FUNCTION_BLOCK FB_GuidanceSystem IMPLEMENTS ITF_HighLevelSystem
VAR_INPUT
	eState : GuidanceSystemSTM;
END_VAR
VAR
	fbAccelerationSensor1 : FB_AccelerationSensor;
	fbAccelerationSensor2 : FB_AccelerationSensor;
	fbGuidanceControllerXMC1 : FB_GuidanceController;
	fbGuidanceControllerXMC2 : FB_GuidanceController;
	fbGuidanceControllerXMC3 : FB_GuidanceController;
	fbGuidanceControllerXMC4 : FB_GuidanceController;
END_VAR

IF eActivationStatus = ActivationStatus.Enabled THEN
	//High Level State Machine
	CASE eState OF
		GuidanceSystemSTM.Idling:
				bEnableCurrentController := FALSE;		

				fbGuidanceControllerXMC1.bActive := FALSE;
				fbGuidanceControllerXMC2.bActive := FALSE;
				fbGuidanceControllerXMC3.bActive := FALSE;
				fbGuidanceControllerXMC4.bActive := FALSE;
		
				fbAccelerationSensor1();
				fbAccelerationSensor2();
				fbGuidanceControllerXMC1();
				fbGuidanceControllerXMC2();
				fbGuidanceControllerXMC3();
				fbGuidanceControllerXMC4();	
		
		
		GuidanceSystemSTM.PreRunning:
				bEnableCurrentController := FALSE;		

				fbAccelerationSensor1();
				fbAccelerationSensor2();
				fbGuidanceControllerXMC1();
				fbGuidanceControllerXMC2();
				fbGuidanceControllerXMC3();
				fbGuidanceControllerXMC4();	
		
		
		GuidanceSystemSTM.Running:
				bEnableCurrentController := TRUE;
		
				fbGuidanceControllerXMC1.bActive := TRUE;
				fbGuidanceControllerXMC2.bActive := TRUE;
				fbGuidanceControllerXMC3.bActive := TRUE;
				fbGuidanceControllerXMC4.bActive := TRUE;

				fbAccelerationSensor1();
				fbAccelerationSensor2();
				fbGuidanceControllerXMC1();
				fbGuidanceControllerXMC2();
				fbGuidanceControllerXMC3();
				fbGuidanceControllerXMC4();		

		GuidanceSystemSTM.PostRunning:
				bEnableCurrentController := FALSE;
		
				fbGuidanceControllerXMC1.bActive := FALSE;
				fbGuidanceControllerXMC2.bActive := FALSE;
				fbGuidanceControllerXMC3.bActive := FALSE;
				fbGuidanceControllerXMC4.bActive := FALSE;
				
				fbAccelerationSensor1();
				fbAccelerationSensor2();
				fbGuidanceControllerXMC1();
				fbGuidanceControllerXMC2();
				fbGuidanceControllerXMC3();
				fbGuidanceControllerXMC4();			
	END_CASE
END_IF

PROPERTY aIMU1Acceleration : ARRAY [0..2] OF REAL
GET
aIMU1Acceleration := fbAccelerationSensor1.aAccelerationValues;
END_GET
END_PROPERTY

PROPERTY aIMU2Acceleration : ARRAY [0..2] OF REAL
GET
aIMU2Acceleration := fbAccelerationSensor1.aAccelerationValues;
END_GET
END_PROPERTY

PROPERTY PUBLIC bEnableCurrentController : BOOL
GET
END_GET
SET // PUBLIC
fbGuidanceControllerXMC1.bActive := bEnableCurrentController;
fbGuidanceControllerXMC2.bActive := bEnableCurrentController;
fbGuidanceControllerXMC3.bActive := bEnableCurrentController;
fbGuidanceControllerXMC4.bActive := bEnableCurrentController;
END_SET
END_PROPERTY

PROPERTY PUBLIC bEnableIControl : BOOL
GET
VAR
	nControlOption : USINT;
END_VAR
nControlOption := nGCControlOption;

IF nControlOption.0 THEN
	bEnableIControl := TRUE;
ELSE
	bEnableIControl := FALSE;
END_IF
END_GET
END_PROPERTY

PROPERTY PUBLIC bEnablePControl : BOOL
GET
VAR
	nControlOption : USINT;
END_VAR
nControlOption := nGCControlOption;

IF nControlOption.1 THEN
	bEnablePControl := TRUE;
ELSE
	bEnablePControl := FALSE;
END_IF
END_GET
END_PROPERTY

PROPERTY eActivationStatus : ActivationStatus
GET
END_GET
SET
END_SET
END_PROPERTY

PROPERTY eCondition : HighLevelCondition
GET
IF eActivationStatus = ActivationStatus.Disabled THEN
	eCondition := HighLevelCondition.SLEEP;
ELSE
	IF fbAccelerationSensor1.eCondition = SubLevelCondition.RUN AND fbAccelerationSensor2.eCondition = SubLevelCondition.RUN AND fbGuidanceController.eCondition = SubLevelCondition.RUN THEN
		eCondition := HighLevelCondition.RUN;
	ELSE
		eCondition := HighLevelCondition.INIT;
	END_IF
END_IF
END_GET
END_PROPERTY

PROPERTY PUBLIC eGCOperationMode : BOOL
SET
IF NOT eGCOperationMode THEN
	fbGuidanceControllerXMC1.eOperationMode := GuidanceControllerOperationMode.CurrentControlled;
	fbGuidanceControllerXMC2.eOperationMode := GuidanceControllerOperationMode.CurrentControlled;
	fbGuidanceControllerXMC3.eOperationMode := GuidanceControllerOperationMode.CurrentControlled;
	fbGuidanceControllerXMC4.eOperationMode := GuidanceControllerOperationMode.CurrentControlled;
ELSE
	fbGuidanceControllerXMC1.eOperationMode := GuidanceControllerOperationMode.ForceControlled;
	fbGuidanceControllerXMC2.eOperationMode := GuidanceControllerOperationMode.ForceControlled;
	fbGuidanceControllerXMC3.eOperationMode := GuidanceControllerOperationMode.ForceControlled;
	fbGuidanceControllerXMC4.eOperationMode := GuidanceControllerOperationMode.ForceControlled;
END_IF
END_SET
END_PROPERTY

PROPERTY PUBLIC fGCAccelerationY : ARRAY [0..3] OF LREAL
SET
fbGuidanceControllerXMC1.fAccelerationY := fGCAccelerationY[0];
fbGuidanceControllerXMC2.fAccelerationY := fGCAccelerationY[1];
fbGuidanceControllerXMC3.fAccelerationY := fGCAccelerationY[2];
fbGuidanceControllerXMC4.fAccelerationY := fGCAccelerationY[3];
END_SET
END_PROPERTY

PROPERTY PUBLIC fGCActualGuidAcceleration : ARRAY [0..3] OF REAL
SET
fbGuidanceControllerXMC1.fActualYAcceleration := fGCActualGuidAcceleration[0];
fbGuidanceControllerXMC2.fActualYAcceleration := fGCActualGuidAcceleration[1];
fbGuidanceControllerXMC3.fActualYAcceleration := fGCActualGuidAcceleration[2];
fbGuidanceControllerXMC4.fActualYAcceleration := fGCActualGuidAcceleration[3];
END_SET
END_PROPERTY

PROPERTY PUBLIC fGCActualGuidCurrent : ARRAY [0..3] OF REAL
SET
fbGuidanceControllerXMC1.fActualCurrent := fGCActualGuidCurrent[0];
fbGuidanceControllerXMC2.fActualCurrent := fGCActualGuidCurrent[1];
fbGuidanceControllerXMC3.fActualCurrent := fGCActualGuidCurrent[2];
fbGuidanceControllerXMC4.fActualCurrent := fGCActualGuidCurrent[3];
END_SET
END_PROPERTY

PROPERTY PUBLIC fGCActualGuidDistance : ARRAY [0..3] OF REAL
SET
fbGuidanceControllerXMC1.fActualYDistance := fGCActualGuidDistance[0];
fbGuidanceControllerXMC2.fActualYDistance := fGCActualGuidDistance[1];
fbGuidanceControllerXMC3.fActualYDistance := fGCActualGuidDistance[2];
fbGuidanceControllerXMC4.fActualYDistance := fGCActualGuidDistance[3];
END_SET
END_PROPERTY

PROPERTY PUBLIC fGCCurrentLeft : ARRAY [0..3] OF LREAL
GET
END_GET
SET
fbGuidanceControllerXMC1.fCurrentLeft := fGCCurrentLeft[0];
fbGuidanceControllerXMC2.fCurrentLeft := fGCCurrentLeft[1];
fbGuidanceControllerXMC3.fCurrentLeft := fGCCurrentLeft[2];
fbGuidanceControllerXMC4.fCurrentLeft := fGCCurrentLeft[3];
END_SET
END_PROPERTY

PROPERTY PUBLIC fGCCurrentRight : ARRAY [0..3] OF LREAL
GET
END_GET
SET
fbGuidanceControllerXMC1.fCurrentRight := fGCCurrentRight[0];
fbGuidanceControllerXMC2.fCurrentRight := fGCCurrentRight[1];
fbGuidanceControllerXMC3.fCurrentRight := fGCCurrentRight[2];
fbGuidanceControllerXMC4.fCurrentRight := fGCCurrentRight[3];
END_SET
END_PROPERTY

PROPERTY PUBLIC fGCDesiredDeviationFromCenterLine : LREAL
GET
END_GET
SET
fbGuidanceControllerXMC1.fDesiredDeviationFromCenterLine := fGCDesiredDeviationFromCenterLine;
fbGuidanceControllerXMC2.fDesiredDeviationFromCenterLine := fGCDesiredDeviationFromCenterLine;
fbGuidanceControllerXMC3.fDesiredDeviationFromCenterLine := fGCDesiredDeviationFromCenterLine;
fbGuidanceControllerXMC4.fDesiredDeviationFromCenterLine := fGCDesiredDeviationFromCenterLine;
END_SET
END_PROPERTY

PROPERTY PUBLIC fGCDistanceLeft1 : ARRAY [0..3] OF LREAL
GET
END_GET
SET
fbGuidanceControllerXMC1.fDistanceLeft1 := fGCDistanceLeft1[0];
fbGuidanceControllerXMC2.fDistanceLeft1 := fGCDistanceLeft1[1];
fbGuidanceControllerXMC3.fDistanceLeft1 := fGCDistanceLeft1[2];
fbGuidanceControllerXMC4.fDistanceLeft1 := fGCDistanceLeft1[3];
END_SET
END_PROPERTY

PROPERTY PUBLIC fGCDistanceLeft2 : ARRAY [0..3] OF LREAL
GET
END_GET
SET
fbGuidanceControllerXMC1.fDistanceLeft2 := fGCDistanceLeft2[0];
fbGuidanceControllerXMC2.fDistanceLeft2 := fGCDistanceLeft2[1];
fbGuidanceControllerXMC3.fDistanceLeft2 := fGCDistanceLeft2[2];
fbGuidanceControllerXMC4.fDistanceLeft2 := fGCDistanceLeft2[3];
END_SET
END_PROPERTY

PROPERTY PUBLIC fGCDistanceRight1 : ARRAY [0..3] OF LREAL
GET
END_GET
SET
fbGuidanceControllerXMC1.fDistanceRight1 := fGCDistanceRight1[0];
fbGuidanceControllerXMC2.fDistanceRight1 := fGCDistanceRight1[1];
fbGuidanceControllerXMC3.fDistanceRight1 := fGCDistanceRight1[2];
fbGuidanceControllerXMC4.fDistanceRight1 := fGCDistanceRight1[3];
END_SET
END_PROPERTY

PROPERTY PUBLIC fGCDistanceRight2 : ARRAY [0..3] OF LREAL
GET
END_GET
SET
fbGuidanceControllerXMC1.fDistanceRight1 := fGCDistanceRight1[0];
fbGuidanceControllerXMC2.fDistanceRight1 := fGCDistanceRight1[1];
fbGuidanceControllerXMC3.fDistanceRight1 := fGCDistanceRight1[2];
fbGuidanceControllerXMC4.fDistanceRight1 := fGCDistanceRight1[3];
END_SET
END_PROPERTY

PROPERTY PUBLIC fGCEstimatedForce : ARRAY [0..3] OF LREAL
GET
END_GET
SET
fbGuidanceControllerXMC1.fEstimatedForce := fGCEstimatedForce[0];
fbGuidanceControllerXMC2.fEstimatedForce := fGCEstimatedForce[1];
fbGuidanceControllerXMC3.fEstimatedForce := fGCEstimatedForce[2];
fbGuidanceControllerXMC4.fEstimatedForce := fGCEstimatedForce[3];
END_SET
END_PROPERTY

PROPERTY PUBLIC fGCOutputGuidCurrent : ARRAY [0..3] OF LREAL
GET
fGCOutputGuidCurrent[0] := fbGuidanceControllerXMC1.fNewReferenceValueForCurrent;
fGCOutputGuidCurrent[1] := fbGuidanceControllerXMC2.fNewReferenceValueForCurrent;
fGCOutputGuidCurrent[2] := fbGuidanceControllerXMC3.fNewReferenceValueForCurrent;
fGCOutputGuidCurrent[3] := fbGuidanceControllerXMC4.fNewReferenceValueForCurrent;
END_GET
END_PROPERTY

PROPERTY PUBLIC fGCOutputGuidForce : ARRAY [0..3] OF LREAL
GET
fGCOutputGuidForce[0] := fbGuidanceControllerXMC1.fNewRefrenceValueForForce;
fGCOutputGuidForce[1] := fbGuidanceControllerXMC2.fNewRefrenceValueForForce;
fGCOutputGuidForce[2] := fbGuidanceControllerXMC3.fNewRefrenceValueForForce;
fGCOutputGuidForce[3] := fbGuidanceControllerXMC4.fNewRefrenceValueForForce;
END_GET
END_PROPERTY

PROPERTY PUBLIC fGCOutputGuidVoltage : ARRAY [0..3] OF LREAL
GET
fGCOutputGuidVoltage[0] := fbGuidanceControllerXMC1.fNewreferenceValueForVoltage;
fGCOutputGuidVoltage[1] := fbGuidanceControllerXMC2.fNewreferenceValueForVoltage;
fGCOutputGuidVoltage[2] := fbGuidanceControllerXMC3.fNewreferenceValueForVoltage;
fGCOutputGuidVoltage[3] := fbGuidanceControllerXMC4.fNewreferenceValueForVoltage;
END_GET
END_PROPERTY

PROPERTY PUBLIC fGCReferenceYSignal : REAL
SET
fbGuidanceControllerXMC1.fDesiredDeviationFromCenterLine := fGCReferenceYSignal;
fbGuidanceControllerXMC2.fDesiredDeviationFromCenterLine := fGCReferenceYSignal;
fbGuidanceControllerXMC3.fDesiredDeviationFromCenterLine := fGCReferenceYSignal;
fbGuidanceControllerXMC4.fDesiredDeviationFromCenterLine := fGCReferenceYSignal;
END_SET
END_PROPERTY

PROPERTY nErrorID : UDINT
GET
VAR
	nErrorBitsIMU1 : UDINT;
	nErrorBitsIMU2 : UDINT;
	nErrorBitsGC : UDINT;
END_VAR
nErrorBitsIMU1 := fbAccelerationSensor1.nErrorID;
nErrorBitsIMU2 := fbAccelerationSensor2.nErrorID;
nErrorBitsGC := fbGuidanceController.nErrorID;

//ErrorBits
nErrorID.0 := nErrorBitsIMU1.0;
nErrorID.1 := nErrorBitsIMU1.1;
nErrorID.2 := nErrorBitsIMU2.0;
nErrorID.3 := nErrorBitsIMU2.1;
nErrorID.4 := nErrorBitsGC.0;
nErrorID.5 := nErrorBitsGC.1;
nErrorID.6 := nErrorBitsGC.2;
nErrorID.7 := nErrorBitsGC.3;
END_GET
END_PROPERTY

PROPERTY PUBLIC nGCControlOption : USINT
SET
IF nGCControlOption.0 THEN
	fbGuidanceControllerXMC1.eOperationMode := GuidanceControllerOperationMode.CurrentControlled;
	fbGuidanceControllerXMC2.eOperationMode := GuidanceControllerOperationMode.CurrentControlled;
	fbGuidanceControllerXMC3.eOperationMode := GuidanceControllerOperationMode.CurrentControlled;
	fbGuidanceControllerXMC4.eOperationMode := GuidanceControllerOperationMode.CurrentControlled;
END_IF

IF nGCControlOption.1 THEN
	fbGuidanceControllerXMC1.eOperationMode := GuidanceControllerOperationMode.ForceControlled;
	fbGuidanceControllerXMC2.eOperationMode := GuidanceControllerOperationMode.ForceControlled;
	fbGuidanceControllerXMC3.eOperationMode := GuidanceControllerOperationMode.ForceControlled;
	fbGuidanceControllerXMC4.eOperationMode := GuidanceControllerOperationMode.ForceControlled;
END_IF
END_SET
END_PROPERTY

END_FUNCTION_BLOCK

(* stored: Version 1.1.0.1, ProductVersion 3.1.4024.12
   POU FB_GuidanceSystem: Id {f33f1b41-c667-4ee8-81c9-ea9b824242db}, SpecialFunc None
   Folder Old: Id {7aa52538-30c4-4cbb-9c21-00f1df212155}
   Property aIMU1Acceleration: Id {d02b525a-bc1b-492a-a816-47305250732e}
   Get Get: Id {a44a823d-8479-4c86-a9d4-e6594c5cc29d}
   Property aIMU2Acceleration: Id {77f151eb-f5be-47a3-8ffb-b31bed26cce9}
   Get Get: Id {dc8e6747-1f97-4ee1-9ae5-87cfe2fd9cb4}
   Property bEnableCurrentController: Id {219914c8-e60f-443e-a9b1-1a8b13359e38}
   Get Get: Id {bf7f780d-3e52-446a-9edc-d33640942d1d}
   Set Set: Id {2f663600-275c-4c09-ac3d-432efceb8dea}
   Property bEnableIControl: Id {283b4a68-da76-43e0-a917-a5beaa4ff21d}
   Get Get: Id {7901ef3c-95bf-4fcd-aea4-a85ff508a55b}
   Property bEnablePControl: Id {bd3c004b-ebc6-4cb2-aa9a-60f50ead2145}
   Get Get: Id {6cf49da1-bee3-4e51-b6b3-b32967b83f0f}
   Property eActivationStatus: Id {7745b1cc-dc82-4592-9cff-4ff71271404b}
   Get Get: Id {d98d84fa-bd91-4902-95be-20e2513aa577}
   Set Set: Id {9ab97794-3bbd-4a17-9257-c2e777c8f634}
   Property eCondition: Id {3adb4534-3e01-4acc-ac7e-71736dcca723}
   Get Get: Id {e8a79d02-6646-46d0-90f1-c5b4226277cf}
   Property eGCOperationMode: Id {a231fff4-af11-4fa6-bbbb-52b81abebd9c}
   Set Set: Id {f0fa56de-d897-454d-9d42-6bb0f2919434}
   Property fGCAccelerationY: Id {5725a796-5fbf-40d8-96ed-3a349b0b33c2}
   Set Set: Id {9ffb675e-b451-48f8-9136-27feee5e4d8a}
   Property fGCActualGuidAcceleration: Id {50ef049f-d04e-4160-aa8f-759304a0e478}
   Set Set: Id {02a9edb8-2f92-4ddd-82ba-d7b8a5f1d6f2}
   Property fGCActualGuidCurrent: Id {d1d75f4c-de5e-4edd-b23c-e2299f3ee5c9}
   Set Set: Id {e897c502-87ea-40ef-a11b-7b58d80912d2}
   Property fGCActualGuidDistance: Id {c4680183-d1f5-4b7e-bfb6-9cc5eec92931}
   Set Set: Id {a3fe579a-6e9f-4932-bb02-d36798227109}
   Property fGCCurrentLeft: Id {53e7dfac-89a9-41bd-8f75-697430052753}
   Get Get: Id {e1527d8e-a7c8-435a-9774-52ee23a137e5}
   Set Set: Id {78ef61bc-7927-46a6-b382-75668327a864}
   Property fGCCurrentRight: Id {f4ace9a4-8882-444c-addb-63ca5db50c0c}
   Get Get: Id {2d6c3067-fe38-40a4-bfab-5d161a7e4e00}
   Set Set: Id {fe97b2ac-675e-4238-ac17-56ccf2282ed3}
   Property fGCDesiredDeviationFromCenterLine: Id {3a201cab-adff-4cdb-ad90-d23f9227f1d6}
   Get Get: Id {3a460340-6e8b-46e9-bef5-daf35ad13318}
   Set Set: Id {cad5b033-edbb-4c78-b405-caac801afd88}
   Property fGCDistanceLeft1: Id {f4927582-b412-4a2e-aad1-e2a9c8857f83}
   Get Get: Id {582a67b4-2150-485a-a261-badb49514447}
   Set Set: Id {a862c4d5-2483-4f85-bf9f-9607a6d7203f}
   Property fGCDistanceLeft2: Id {387f246a-be57-4749-8e34-4bf07a8c5edf}
   Get Get: Id {9e3b80c5-cc02-4194-a918-1c445527da47}
   Set Set: Id {3d8abd82-3e87-43b5-986f-94a1b474b5ad}
   Property fGCDistanceRight1: Id {2f668c60-f489-47b4-9a52-93344ff7ef5e}
   Get Get: Id {209f9647-81c7-4875-a451-5a0898bc2858}
   Set Set: Id {2bee9565-beca-4c09-a94e-dceb262c36bd}
   Property fGCDistanceRight2: Id {a054a12f-fdb1-496d-8f54-16db3cfeaca9}
   Get Get: Id {1e70c775-2cf9-431b-843a-34ee340222d5}
   Set Set: Id {41235b03-1187-47eb-8ee5-54e7694adf4d}
   Property fGCEstimatedForce: Id {b081ce65-2e2f-4a44-a910-47e503c93926}
   Get Get: Id {c859e7b8-de91-4b93-89e1-891e1f2e935b}
   Set Set: Id {5c85c87e-7f2f-47b5-9f9d-4e9145e30e4a}
   Property fGCOutputGuidCurrent: Id {f9b9b387-cd33-4a0c-9051-187e4861c041}
   Get Get: Id {658df739-eac8-4c06-8550-f0a57655a7e1}
   Property fGCOutputGuidForce: Id {6807a8ec-a68a-4f62-83c5-b1875dd50002}
   Get Get: Id {b1e1e70e-496f-4e91-a07a-580c756b018f}
   Property fGCOutputGuidVoltage: Id {786a695b-7ef5-4e4b-9a0a-d28af41c4a96}
   Get Get: Id {a13fbcfd-83c0-48f5-9cc8-d5358855f974}
   Property fGCReferenceYSignal: Id {315060d2-d961-478e-ab2d-1c6a1e6d7fef}
   Set Set: Id {22b21363-0bc6-4c27-96bd-13c3bba80b3f}
   Property nErrorID: Id {2b44044c-3e52-4895-8a43-413a23ecd304}
   Get Get: Id {4e75dc01-1205-4771-a577-916f014dc2dc}
   Property nGCControlOption: Id {b651e7a8-a4e6-441f-9f9b-735901e3547d}
   Set Set: Id {3cccd4eb-b1c2-4aad-a797-85ea078b3414} *)
